(* IEC 61131-3 sources: plc_generation_empirical_study/datasets/packages/internal_v0_1_precalibration_20260810/public_tasks/C04_H01_qualified_event_counter, 1 file *)

(* ---- interface.st ---- *)
FUNCTION_BLOCK C04_H01_qualified_event_counter
VAR_INPUT
    Event : BOOL;
    Qualify : BOOL;
    Reset : BOOL;
    Limit : INT;
END_VAR
VAR_OUTPUT
    Count : INT;
    AcceptedPulse : BOOL;
    AtLimit : BOOL;
END_VAR
END_FUNCTION_BLOCK
